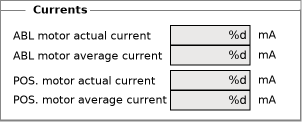
VISUALIZATION VISU_M3RotationCurrents  // 302x122
VAR_IN_OUT
	ref : M3Rotation;
    widget : M3RotationWidget;
END_VAR
    Label (10,71 195x20), "POS. motor actual current"
    Label (255,70 35x20), "mA"
    Rectangle (170,70 80x20), "%d", text variable: ref.parts.positioningDrive.actualCurrent.milliAmps.value
    Label (10,26 190x20), "ABL motor actual current"
    Label (255,25 35x20), "mA"
    Rectangle (170,25 80x20), "%d", text variable: ref.parts.antiBacklashDrive.actualCurrent.milliAmps.value
    Label (10,46 190x20), "ABL motor average current"
    Label (255,45 35x20), "mA"
    Rectangle (170,45 80x20), "%d", text variable: ref.parts.antiBacklashDrive.averageCurrent.milliAmps.value
    Label (255,90 35x20), "mA"
    Rectangle (170,90 80x20), "%d", text variable: ref.parts.positioningDrive.averageCurrent.milliAmps.value
    Label (10,90 195x20), "POS. motor average current"
    Label (30,0 150x20), "Currents"
    Polyline (90,10) (300,10) (300,120) (0,120) (0,10) (25,10)
END_VISUALIZATION

(* stored: Version 1.1.0.1, ProductVersion 3.1.4018.2
   Visu VISU_M3RotationCurrents: Id {a1b39729-7c9b-4765-a6ae-9a97be33572c} *)
